FUNCTION TryConvert_WORD_TO_DT : BOOL
VAR_INPUT
	in : WORD;
	out : REFERENCE TO DT;
END_VAR

out := WORD_TO_DT(in);
TryConvert_WORD_TO_DT := TRUE;

END_FUNCTION

(* stored: Version 1.1.0.1, ProductVersion 3.1.4024.12
   POU TryConvert_WORD_TO_DT: Id {6df3fc83-4a7d-4ad4-bf1c-6be2c737e414}, SpecialFunc None *)
